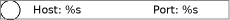
VISUALIZATION _VISU_CameraTcpIpSetting  // 230x20
VAR_IN_OUT
	m_Inst : FB_CameraTcpIp;
END_VAR
    Ellipse (0,0 20x20)
        toggle m_Inst._pFbTcpIpClient^.bEnable
    Rectangle (30,0 120x20), "Host: %s", tooltip "Camera ip address", text variable: m_Inst._pFbTcpIpClient^.sRemoteHost
    Rectangle (150,0 80x20), "Port: %s", tooltip "camera port", text variable: m_Inst._pFbTcpIpClient^.nRemotePort
END_VISUALIZATION

(* stored: Version 1.1.0.1, ProductVersion 3.1.4024.3
   Visu _VISU_CameraTcpIpSetting: Id {38f3200e-af91-4373-a779-1e9595a37d59} *)
